FUNCTION_BLOCK Model (* Composite Function Block Type *)
  (* Standard: 61499-2 *)
  (* Version 0.0, 7/13/2016, Andrei, nxtControl GmbH, template *)
  PACKAGE Main;
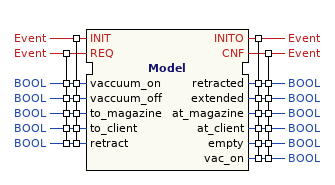
  EVENT_INPUT
    INIT WITH retract, to_magazine, to_client, vaccuum_off, vaccuum_on; (* Initialization Request *)
    REQ WITH retract, to_magazine, to_client, vaccuum_off, vaccuum_on; (* Normal Execution Request *)
  END_EVENT
  EVENT_OUTPUT
    INITO WITH extended, retracted, at_magazine, at_client, vac_on, empty; (* Initialization Confirm *)
    CNF WITH extended, retracted, at_magazine, at_client, vac_on, empty; (* Execution Confirmation *)
  END_EVENT
  VAR_INPUT
    vaccuum_on : BOOL;
    vaccuum_off : BOOL;
    to_magazine : BOOL;
    to_client : BOOL;
    retract : BOOL; (* Input event qualifier *)
  END_VAR
  VAR_OUTPUT
    retracted : BOOL;
    extended : BOOL; (* Output event qualifier *)
    at_magazine : BOOL;
    at_client : BOOL;
    empty : BOOL;
    vac_on : BOOL;
  END_VAR
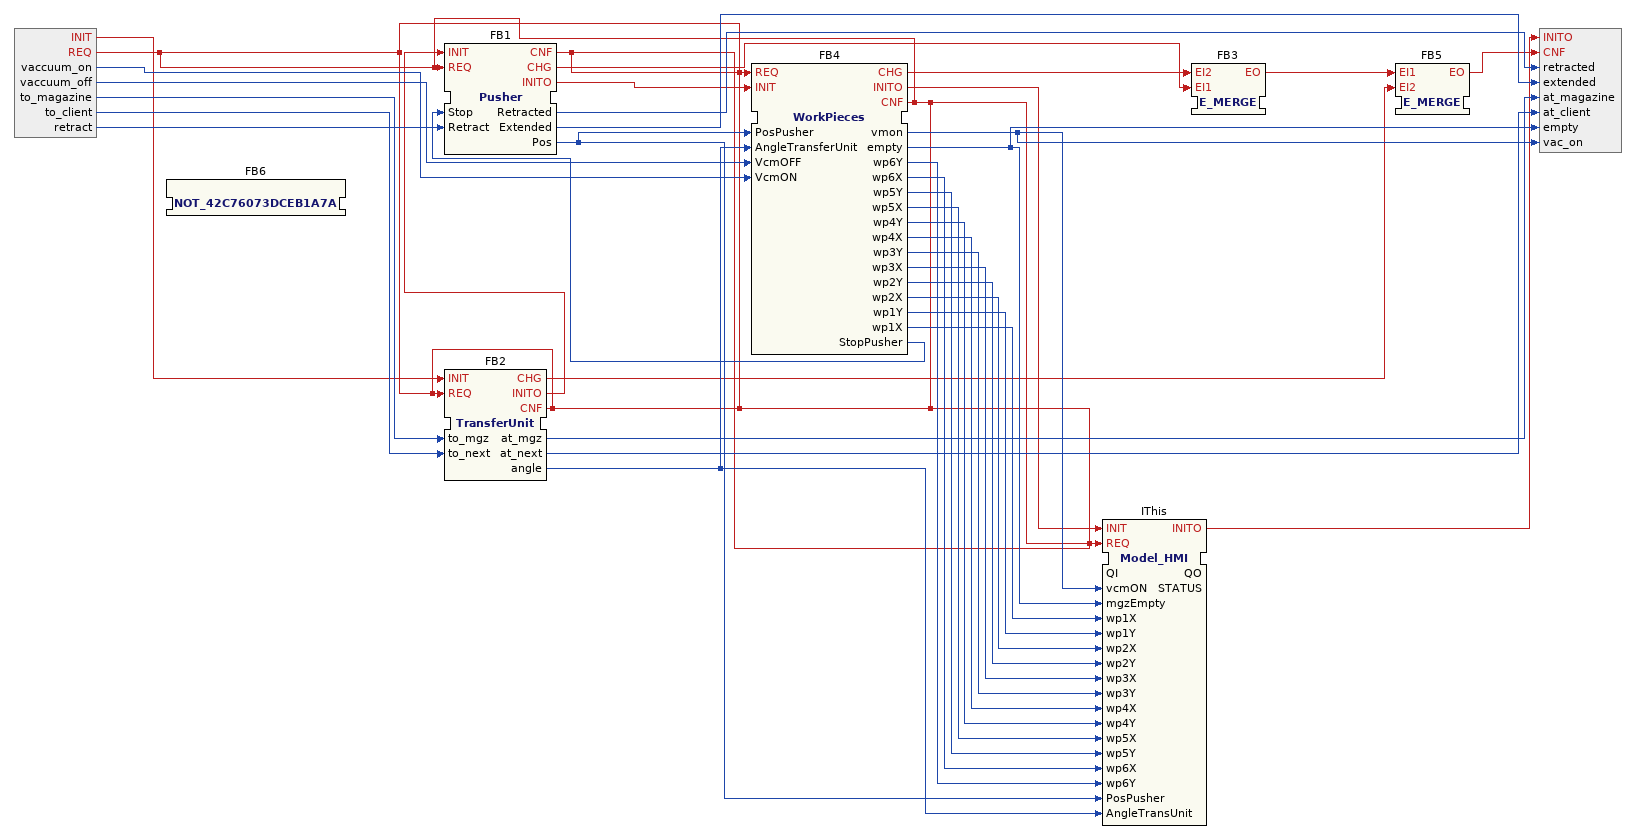
  FBS
    FB3 : E_MERGE;
    FB5 : E_MERGE;
    FB2 : TransferUnit;
    FB4 : WorkPieces;
    IThis : Model_HMI;
    FB1 : Pusher;
    FB6 : NOT_42C76073DCEB1A7A; {SET_ATTRIBUTE(Configuration.GenericFBType.InterfaceParams, Runtime.Standard#CNT:=1;OUT${CNT$}:BOOL)}
  END_FBS
  EVENT_CONNECTIONS
    FB1.CNF TO FB4.REQ;
    FB4.CHG TO FB3.EI2;
    FB1.CHG TO FB3.EI1;
    FB3.EO TO FB5.EI1;
    FB2.CHG TO FB5.EI2;
    FB2.INITO TO FB1.INIT;
    INIT TO FB2.INIT;
    REQ TO FB1.REQ;
    REQ TO FB2.REQ;
    FB1.INITO TO FB4.INIT;
    FB2.CNF TO FB4.REQ;
    FB5.EO TO CNF;
    IThis.INITO TO INITO;
    FB4.INITO TO IThis.INIT;
    FB4.CNF TO IThis.REQ;
    FB2.CNF TO IThis.REQ;
    FB1.CNF TO IThis.REQ;
    REQ TO FB4.REQ;
    FB4.CNF TO FB1.REQ;
    FB4.CNF TO FB2.REQ;
  END_CONNECTIONS
  DATA_CONNECTIONS
    to_magazine TO FB2.to_mgz;
    to_client TO FB2.to_next;
    FB2.at_mgz TO at_magazine;
    FB2.at_next TO at_client;
    FB1.Retracted TO retracted;
    FB1.Extended TO extended;
    FB1.Pos TO FB4.PosPusher;
    FB2.angle TO FB4.AngleTransferUnit;
    FB4.vmon TO vac_on;
    FB4.empty TO empty;
    FB2.angle TO IThis.AngleTransUnit;
    FB1.Pos TO IThis.PosPusher;
    FB4.wp6Y TO IThis.wp6Y;
    FB4.wp6X TO IThis.wp6X;
    FB4.wp5Y TO IThis.wp5Y;
    FB4.wp5X TO IThis.wp5X;
    FB4.wp4Y TO IThis.wp4Y;
    FB4.wp4X TO IThis.wp4X;
    FB4.wp3Y TO IThis.wp3Y;
    FB4.wp3X TO IThis.wp3X;
    FB4.wp2Y TO IThis.wp2Y;
    FB4.wp2X TO IThis.wp2X;
    FB4.wp1Y TO IThis.wp1Y;
    FB4.wp1X TO IThis.wp1X;
    FB4.StopPusher TO FB1.Stop;
    FB4.vmon TO IThis.vcmON;
    FB4.empty TO IThis.mgzEmpty;
    retract TO FB1.Retract;
    vaccuum_off TO FB4.VcmOFF;
    vaccuum_on TO FB4.VcmON;
  END_CONNECTIONS
END_FUNCTION_BLOCK
